Staubli VAL3: get.pgx

public program get(string& x_sItem[], num x_nIndex)
begin
  //
  // get one element from the list
  //
end
